PROGRAM P_Demo_EIB_BIT_SEND_EX
VAR
    fbEIB_BIT_SEND_EX         : EIB_BIT_SEND_EX;
    stEibRec            : EIB_REC;
    stGroup             : EIB_GROUP_ADDR := (MAIN := 1, SUB_MAIN := 1, NUMBER := 50);
    bSendStart          : BOOL;
    iWorkMode           : INT := 3;
    tCyclePeriod        : TIME := T#5S;
    tMinIntervalChange  : TIME := T#500MS;
    data                : BOOL := FALSE;
    bResponseToRead     : BOOL := TRUE;
    bSendBusy           : BOOL;
    bSendError          : BOOL;
    iLastErrID          : EIB_ERROR_CODE;
END_VAR

// ============================================================
// Tc2_EIB.EIB_BIT_SEND_EX 演示程序
// ============================================================
// 场景：PLC 开关命令发送到 EIB 组 1/1/50，模式 OnChangePolling：心跳 + 即时变化 + 响应 read。
// 价值：周期心跳 + 即时变化 + 主动答查；BMS 工程首选
// 验证步骤：
//   1. 右键 PLC 项目下 POUs 文件夹 → Add → Existing Item → 选本 .TcPOU 文件
//   2. 引用 Tc2_EIB（References → Add library）
//   3. 编译 → 登录 → 运行；按下方在线写值步骤操作
// 验证：登录 `bSendStart := TRUE` → 周期 5 秒看到 1/1/50 出帧；改 data 立即出帧。
// ============================================================

fbEIB_BIT_SEND_EX(
    bStart         := bSendStart,
    iMode          := iWorkMode,
    CyclePolling   := tCyclePeriod,
    MinSendTime    := tMinIntervalChange,
    Group_Address  := stGroup,
    bData          := data,
    str_Rec        := stEibRec,
    bEnableReadReq := bResponseToRead,
    bBusy          => bSendBusy,
    bError         => bSendError,
    iErrorID       => iLastErrID
);

END_PROGRAM

(* stored: Version 1.1.0.1, ProductVersion 3.1.4024.5
   POU P_Demo_EIB_BIT_SEND_EX: Id {2c1a9fb6-f780-5134-a080-3eb104036412}, SpecialFunc None *)
